Omron Sysmac Studio project node_red (Sysmac Studio 1.47.0.64008, StandardProject)

# Controller new_Controller_0: NX1P2-9024DT version 1.40
Task PrimaryTask (priority 4, period or condition 2000): Program0

VAR_GLOBAL RETAIN
    SETPOINT AT %D5 : INT;  (* published *)
    A1 AT %D7 : INT;  (* published *)
    VALUE AT %D8 : INT;
END_VAR

PROGRAM Program0
VAR
    Timer_1 : BOOL;
    timer_a1 : TON;
    T : TIME;
    C : INT;
END_VAR
VAR_EXTERNAL
    A1 : INT;
    VALUE : INT;
    SETPOINT : INT;
END_VAR
VAR
    _e1 : R_TRIG;
END_VAR

(* Section Section0: ladder, written here as Structured Text *)

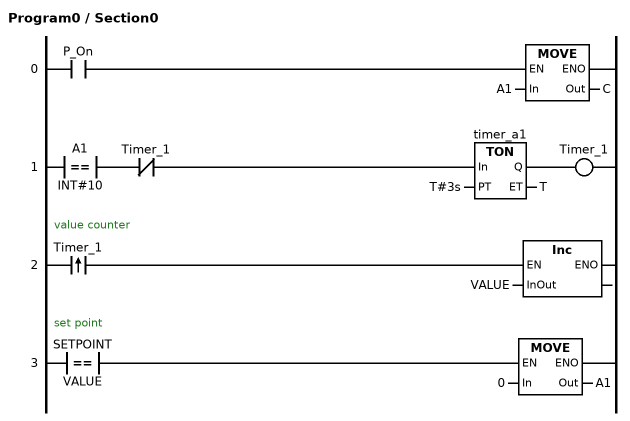
(* Rung 0 *)
IF P_On THEN C := A1; END_IF;
(* Rung 1 *)
timer_a1(In := (A1 = INT#10) AND NOT Timer_1, PT := T#3s, ET => T);
Timer_1 := timer_a1.Q;
(* Rung 2: value counter *)
_e1(CLK := Timer_1);
IF _e1.Q THEN Inc(InOut := VALUE); END_IF;
(* Rung 3: set point *)
IF SETPOINT = VALUE THEN A1 := 0; END_IF;
END_PROGRAM